// TIA Portal V17 export
// export: Created 2022-07-20T06:59:39.9459073Z, ExportSetting WithDefaults, DisplayName Totally Integrated Automation Portal, DisplayVersion V17, DisplayName TIA Portal Openness, DisplayVersion V17, DisplayName TIA Portal Version Control Interface, DisplayVersion V17, DisplayName SINAMICS Startdrive Advanced, DisplayVersion V17, DisplayName SINAMICS Startdrive G130, G150, S120, S150, SINAMICS MV, S210, DisplayVersion V17, DisplayName SINAMICS Startdrive G110M, G120, G120C, G120D, G120P, G115D, DisplayVersion V17, DisplayName STEP 7 Professional, DisplayVersion V17, DisplayName STEP 7 Safety, DisplayVersion V17, DisplayName WinCC Advanced, DisplayVersion V17
FUNCTION "FC10018_DateToString" : String   // FC10018, LAD
{ S7_Optimized_Access := 'TRUE' }
VERSION : 0.1
// stored: AutoNumber false, IsIECCheckEnabled false, SetENOAutomatically false, UDAEnableTagReadback false
   VAR_INPUT
      DTL_In : DTL;
   END_VAR
BEGIN

REGION Network 1 (SCL): DTL To String Conversion Management
   #FC10018_DateToString := CONCAT(IN1 := DELETE(IN := USINT_TO_STRING(#DTL_In.DAY), L := 1, P := 1),
                                   IN2 := '-',
                                   IN3 := DELETE(IN := USINT_TO_STRING(#DTL_In.MONTH), L := 1, P := 1),
                                   IN4 := '-',
                                   IN5 := DELETE(IN := UINT_TO_STRING(#DTL_In.YEAR), L := 1, P := 1),
                                   IN6 := ' ',
                                   IN7 := DELETE(IN := USINT_TO_STRING(#DTL_In.HOUR), L := 1, P := 1),
                                   IN8 := ':',
                                   IN9 := DELETE(IN := USINT_TO_STRING(#DTL_In.MINUTE), L := 1, P := 1),
                                   IN10 := ':',
                                   IN11 := DELETE(IN := USINT_TO_STRING(#DTL_In.SECOND), L := 1, P := 1),
                                   IN12 := ':',
                                   IN13 := DELETE(IN := UDINT_TO_STRING(#DTL_In.NANOSECOND / 1000000), L := 1, P := 1));
END_REGION
END_FUNCTION
